(*

.. <legal notes>

legal notes
=================
| SPDX-FileCopyrightText: © 2026 Oleksandr Tiutyk <trofimich@gmail.com>
| SPDX-License-Identifier: LGPL-3.0-only
| For details check: LGPL-3.0-only_

.. _LGPL-3.0-only: https://www.gnu.org/licenses/lgpl-3.0.en.html

.. </legal notes>

*)

{attribute 'no_explicit_call' := 'Direct call is not allowed'} 
FUNCTION_BLOCK ABSTRACT Object IMPLEMENTS IObject

{attribute 'monitoring' := 'call'}
PROPERTY ABSTRACT ClassName : STRING
GET
END_GET
END_PROPERTY

{attribute "object_name" := "Equals"}
METHOD Equals : BOOL
VAR_INPUT 
	object : IObject;
END_VAR
VAR
	selfPointer : POINTER TO Object;
	comparingPointer : POINTER TO Object;
END_VAR
selfPointer := THIS;

IF __QUERYPOINTER(object, comparingPointer) THEN
	Equals := selfPointer = comparingPointer;
END_IF
END_METHOD

METHOD FB_exit : BOOL
VAR_INPUT
	bInCopyCode : BOOL; // if TRUE, the exit method is called for exiting an instance that is copied afterwards (online change).
END_VAR
IF ObjectStatisticsSettings.CountObjectStatistics THEN
	ObjectStatistics.RemoveObject(THIS^);
END_IF
END_METHOD

METHOD FB_init : BOOL
VAR_INPUT
	bInitRetains : BOOL; // if TRUE, the retain variables are initialized (warm start / cold start)
	bInCopyCode : BOOL; // if TRUE, the instance afterwards gets moved into the copy code (online change)
END_VAR
IF ObjectStatisticsSettings.CountObjectStatistics THEN
	ObjectStatistics.AddObject(THIS^);
END_IF
END_METHOD

METHOD PROTECTED FINAL GetDefaultName : WSTRING
GetDefaultName := TO_WSTRING(Strings.Concat255(ClassName, ' (0x', Tc2_Utilities.LWORD_TO_HEXSTR(TO_LWORD(THIS), 16, FALSE), ')'));
END_METHOD

METHOD GetName : WSTRING
VAR
	named : INamed;
END_VAR
IF __QUERYINTERFACE(THIS^, named) THEN
	GetName := named.Name;
ELSE
	GetName := GetDefaultName();
END_IF
END_METHOD

{attribute 'monitoring' := 'call'}
PROPERTY FINAL IsDynamicInstance : BOOL
GET
IsDynamicInstance := Memory.IsDynamicData(THIS, 1);
END_GET
END_PROPERTY

{attribute 'monitoring' := 'call'}
PROPERTY ABSTRACT NamespaceName : STRING
GET
END_GET
END_PROPERTY

{attribute 'monitoring' := 'call'}
PROPERTY FINAL SelfAddress : POINTER TO Object
GET
SelfAddress := THIS;
END_GET
END_PROPERTY

{attribute 'monitoring' := 'call'}
PROPERTY ABSTRACT SelfSize : ULINT
GET
END_GET
END_PROPERTY

// Returns a string representation of the object for debugging and logging purposes.
// It is recommended to include key properties in a human-readable format.
METHOD ToLogString : WSTRING(255)
VAR_INST
	cachedResult : WSTRING(255);
END_VAR
IF cachedResult = "" THEN
	WideStrings.AppendToTarget255(cachedResult, TO_WSTRING(NamespaceName), ".", TO_WSTRING(ClassName));
END_IF 

ToLogString := cachedResult;
END_METHOD

END_FUNCTION_BLOCK

(* stored: Version 1.1.0.1
   POU Object: Id {65208310-8b3f-466c-81b7-6cce45022676}, SpecialFunc None
   Folder Service members: Id {f442a49f-4b06-4aa2-85a7-5f5794dfab20}
   Property ClassName: Id {93bace28-41b5-44d6-b854-9ee3edbd382f}
   Get Get: Id {64b538df-f61f-4f5f-95f8-f82623c92e0a}
   Method Equals: Id {c147fb9a-ab41-452b-8012-567d8446205b}
   Method FB_exit: Id {2d9f8d8d-3924-4b67-aafc-98d5a0623fe6}
   Method FB_init: Id {f1b8d6f4-27df-492c-b43a-c682b4e0f7b2}
   Method GetDefaultName: Id {3ae22fad-cdcc-4ba8-a264-9144f84c2553}
   Method GetName: Id {257730f6-dd97-4461-8e3a-d2666d17bc44}
   Property IsDynamicInstance: Id {24998a7a-78a1-4ed7-9b02-1f1a03f8b719}
   Get Get: Id {13a65fb5-a1f5-4c18-8711-a901f8b8c50f}
   Property NamespaceName: Id {c3b0678c-30f0-404d-91d4-2a5aabe2e5cc}
   Get Get: Id {816ff93c-7d0c-4e8e-8788-09a43eca472a}
   Property SelfAddress: Id {fb693a32-9773-4047-aa8f-22abdeeaa290}
   Get Get: Id {9f8bbfa3-aa5e-447f-898b-426110e9c9ed}
   Property SelfSize: Id {e1435e8d-7dee-46fb-af88-e0c12efed32f}
   Get Get: Id {6e225585-3ad3-46c5-8df1-c249905d905a}
   Method ToLogString: Id {0a892b58-fb3d-4452-8b29-2d0341433629} *)
